Staubli VAL3: onStart.pgx

program onStart()
  local num i
  local string l_sPath
begin
  // define the page
  cls()
  // set small wiew
  bLarge=false
  bPage=false
  bShowInit=false
  // INIT the resource
  use:bUseRefresh=true
  logMsg("[KERNEL] INTERFACE:PAGE Production")
end
